Fanuc TP program (LS listing): home.ls

/PROG  HOME
/ATTR
OWNER		= MNEDITOR;
COMMENT		= "";
PROG_SIZE	= 206;
CREATE		= DATE 19-04-18  TIME 15:54:38;
MODIFIED	= DATE 19-04-18  TIME 15:55:18;
FILE_NAME	= ;
VERSION		= 0;
LINE_COUNT	= 7;
MEMORY_SIZE	= 550;
PROTECT		= READ_WRITE;
TCD:  STACK_SIZE	= 0,
      TASK_PRIORITY	= 50,
      TIME_SLICE	= 0,
      BUSY_LAMP_OFF	= 0,
      ABORT_REQUEST	= 0,
      PAUSE_REQUEST	= 0;
DEFAULT_GROUP	= 1,*,*,*,*;
CONTROL_CODE	= 00000000 00000000;
/MN
   1:  UTOOL_NUM=1 ;
   2:  UFRAME_NUM=12 ;
   3:   ;
   4:J PR[1:HOME] 100% CNT100    ;
   5:   ;
   6:   ;
   7:   ;
/POS
/END
